Yaskawa INFORM job: HOME-POSITION-ROBOT.JBI

/JOB
//NAME HOME-POSITION-ROBOT
//POS
///NPOS 0,0,0,1,0,0
///TOOL 0
///POSTYPE PULSE
///PULSE
P00000=0,-222014,-26224,0,-132993,0
//INST
///DATE 2018/11/01 12:37
///ATTR SC,RW
///GROUP1 RB1
NOP
MOVJ P0000 VJ=15.00
WAIT SOUT#(57)=ON
SETREG MREG#(1) 1
TIMER T=1.00
END
